RoboDK station: Origenes_adicionales.rdk

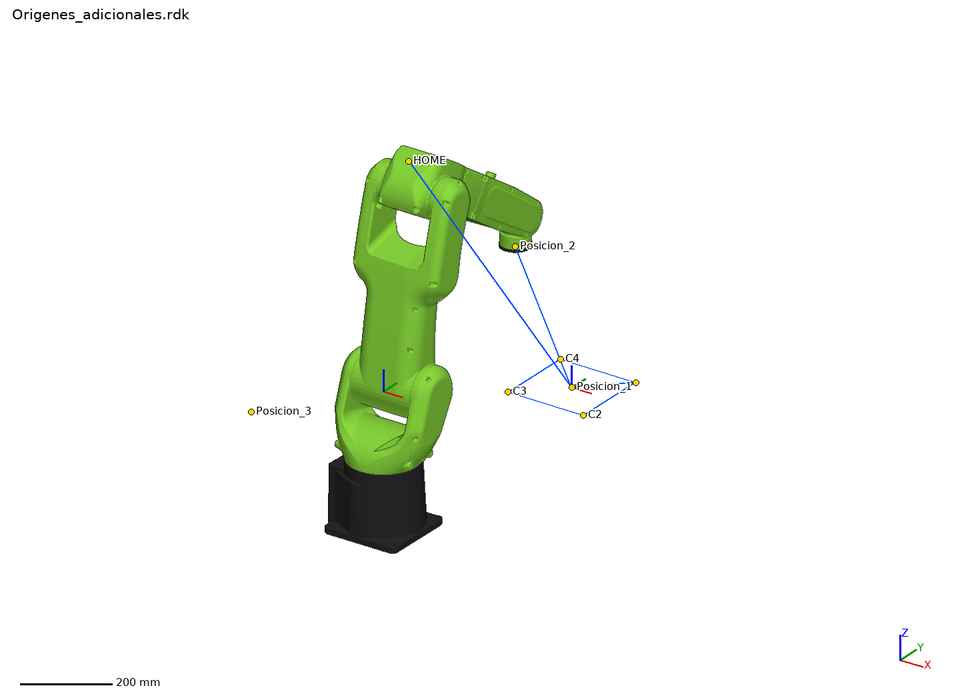
[picture v0: the station drawn from its stored meshes, robots at their saved joint values, targets as dots, program paths as lines]
Station Origenes_adicionales (saved by RoboDK 5.8.0). Poses are relative to the parent item; angles as X-Y-Z fixed-axis rotations.
  - frame Fanuc CR-7iA/L Base at (0, 0, 330) mm
    - robot Fanuc CR-7iA/L: 6 axes, payload 7 kg, reach 911 mm, repeatability 0.03 mm, weight 55 kg
        modified DH rows (alpha deg, a mm, theta deg, d mm): 0, 0, 0, 330; -90, 50, -90, 0; 0, 440, 0, 0; -90, 35, 0, 420; 90, 0, 0, 0; -90, 0, 0, 80
        base shift (0, 0, -330) mm
        joint limits [-170, -100, -67, -190, -115, -360] to [170, 145, 213, 190, 115, 360]; home [0, 0, 0, 0, 0, 0]; saved at [90, 10.532, -33.494, 0, -56.506, -90]
    - target HOME (Cartesian target) at (67.68, 0, 576.29) mm, rotated rx -180 ry -45 rz 0 deg; joints [0, -45, 45, 0, -90, 0] of Fanuc CR-7iA/L
    - target Posicion_1 (Cartesian target) at (500, 0, 150) mm, rotated rx -180 ry 0 rz 0 deg; joints [0, 10.532, -33.494, 0, -56.506, 0] of Fanuc CR-7iA/L
    - target Posicion_2 (Cartesian target) at (0, 500, 150) mm, rotated rx -180 ry 0 rz 0 deg; joints [90, 10.532, -33.494, 0, -56.506, -90] of Fanuc CR-7iA/L
    - target Posicion_3 (Cartesian target) at (0, -500, 150) mm, rotated rx -180 ry 0 rz 0 deg; joints [-90, 10.532, -33.494, 0, -56.506, 90] of Fanuc CR-7iA/L
  - frame Referencia_1 at (500, 0, 480) mm
    - target C1 (Cartesian target) at (100, 100, 0) mm, rotated rx -180 ry 0 rz 0 deg; joints [9.462, 23.351, -29.142, 0, -60.858, -9.462] of Fanuc CR-7iA/L
    - target C2 (Cartesian target) at (100, -100, 0) mm, rotated rx -180 ry 0 rz 0 deg; joints [-9.462, 23.351, -29.142, 0, -60.858, 9.462] of Fanuc CR-7iA/L
    - target C3 (Cartesian target) at (-100, -100, 0) mm, rotated rx -180 ry 0 rz 0 deg; joints [-14.036, -0.405, -34.648, 0, -55.352, 14.036] of Fanuc CR-7iA/L
    - target C4 (Cartesian target) at (-100, 100, 0) mm, rotated rx -180 ry 0 rz 0 deg; joints [14.036, -0.405, -34.648, 0, -55.352, -14.036] of Fanuc CR-7iA/L
  - program main (12 instructions, listed below)
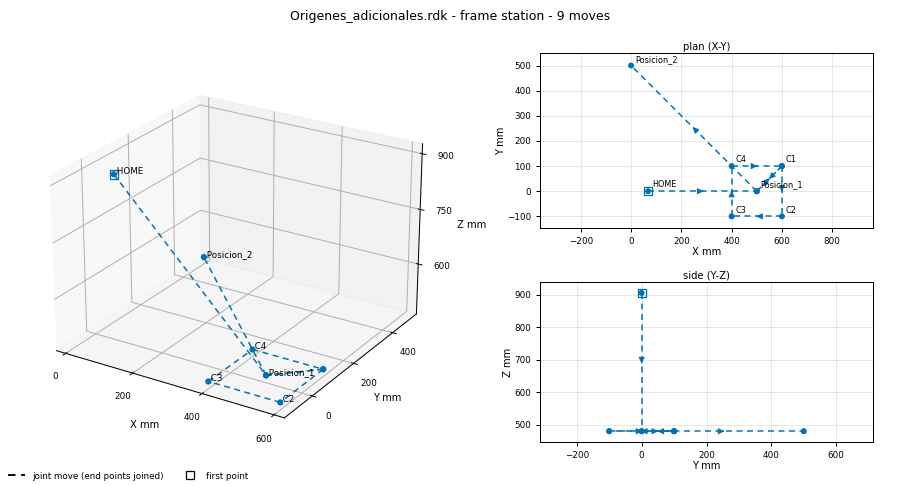
[picture p0: tool path of Origenes_adicionales.rdk in frame station, 9 of 9 moves have a stored position in this frame; points joined in program order, loops and branches not executed]

--- program main (robot Fanuc CR-7iA/L) ---
  Est. Ref.: Fanuc CR-7iA/L Base
  MoveJ (HOME)
  MoveJ (Posicion_1)
  Est. Ref.: Referencia_1
  MoveJ (C1)
  MoveJ (C2)
  MoveJ (C3)
  MoveJ (C4)
  MoveJ (C1)
  Est. Ref.: Fanuc CR-7iA/L Base
  MoveJ (Posicion_1)
  MoveJ (Posicion_2)
